// TIA Portal V19 export
VAR_GLOBAL   // PLC tag table "U2Em4_Output"
   gripperCylinderWorkPositionU2Em4_3 AT %Q182.4 : Bool;   // U2Em4_gripper cylinder 3 working position / Em130_夹爪气缸3工作位
   gripperCylinderWorkPositionU2Em4_4 AT %Q182.6 : Bool;   // U2Em4_gripper cylinder 4 working position / Em130_夹爪气缸4工作位
   gripperCylinderHomePositionU2Em4_2 AT %Q182.3 : Bool;   // U2Em4_Jaw Cylinder 2 Home Position / Em130_夹爪气缸2原位
   gripperCylinderHomePositionU2Em4_3 AT %Q182.5 : Bool;   // U2Em4_Jaw Cylinder 3 Home Position / Em130_夹爪气缸3原位
   gripperCylinderHomePositionU2Em4_1 AT %Q182.1 : Bool;   // U2Em4_Jaw Cylinder 1 Home Position / Em130_夹爪气缸1原位
   gripperCylinderWorkPositionU2Em4_2 AT %Q182.2 : Bool;   // U2Em4_gripper cylinder 2 working position / Em130_夹爪气缸2工作位
   gripperCylinderHomePositionU2Em4_4 AT %Q182.7 : Bool;   // U2Em4_Jaw Cylinder 4 Home Position / Em130_夹爪气缸4原位
   gripperCylinderWorkPositionU2Em4_1 AT %Q182.0 : Bool;   // U2Em4_gripper cylinder 1 working position / Em130_夹爪气缸1工作位
END_VAR
